# EPICS autosave request: NDFileRaw_settings.req
file "NDPluginFile_settings.req", P=$(P), R=$(R)
